// TIA Portal V21 export
FUNCTION_BLOCK "DigitalOutput"   // FB4, LAD
TITLE = FB4
{ S7_Optimized_Access := 'FALSE' }
// DIGITAL OUTPUT
// stored: AutoNumber false, SetENOAutomatically false
   VAR_INPUT
      Cmd { ExternalVisible := 'False'} : Bool;
      SimulationOn { ExternalVisible := 'False'} : Bool;
      MotorFeedbackInputSelection { ExternalVisible := 'False'} : Bool;
      MotorFeedbackInput { ExternalVisible := 'False'} : Bool;
      WaterSensorSelection { ExternalVisible := 'False'} : Bool;
      WaterSensorInput { ExternalVisible := 'False'} : Bool;
      AlwaysTrue : Bool;
      AlwaysFalse : Bool;
      OpenClose : Bool;   // For Valve Only
      Spare_3 : Bool;   // For Valve Only
      ValveFeedbackInputSelection { ExternalVisible := 'False'} : Bool;
      ValveFeedbackInput { ExternalVisible := 'False'} : Bool;
      Interlock : Bool;
      FBCheckDelay { ExternalVisible := 'False'} : Int;
      WSCheckDelay { ExternalVisible := 'False'} : Int;
      secs { ExternalVisible := 'False'} : Bool;
      AlarmAck { ExternalVisible := 'False'} : Bool;
      ModeSel : Bool;   // 1=Man/ 0=Auto
      Fault : Bool;
      Reset : Bool;
      spare : Bool;
      spare_1 : Bool;
      spare_2 : Bool;
   END_VAR
   VAR_OUTPUT
      Output { ExternalVisible := 'False'} : Bool;
      FeedBackTripAlarm : Bool;
      NoWaterFlowAlarm : Bool;
      LineColour : DInt;
      ValveColour : DInt;
      Mode : DInt;   // Auto=0 , Manual=1
      Status : DInt;
   END_VAR
   VAR_IN_OUT
      OpFbTrip { ExternalVisible := 'False'} : Bool;
      OpWaterSensorTrip { ExternalVisible := 'False'} : Bool;
      FBCheckActualTime { ExternalVisible := 'False'} : Int;
      WSCheckActualTime { ExternalVisible := 'False'} : Int;
   END_VAR
   VAR
      ResetBtn { S7_SetPoint := 'True'} : TON_TIME;
   END_VAR
   VAR_TEMP   // added for the SCL form of the ladder/FBD networks
      _w1 : Bool;
      _w2 : Bool;
   END_VAR
BEGIN

REGION Network 1: #Output
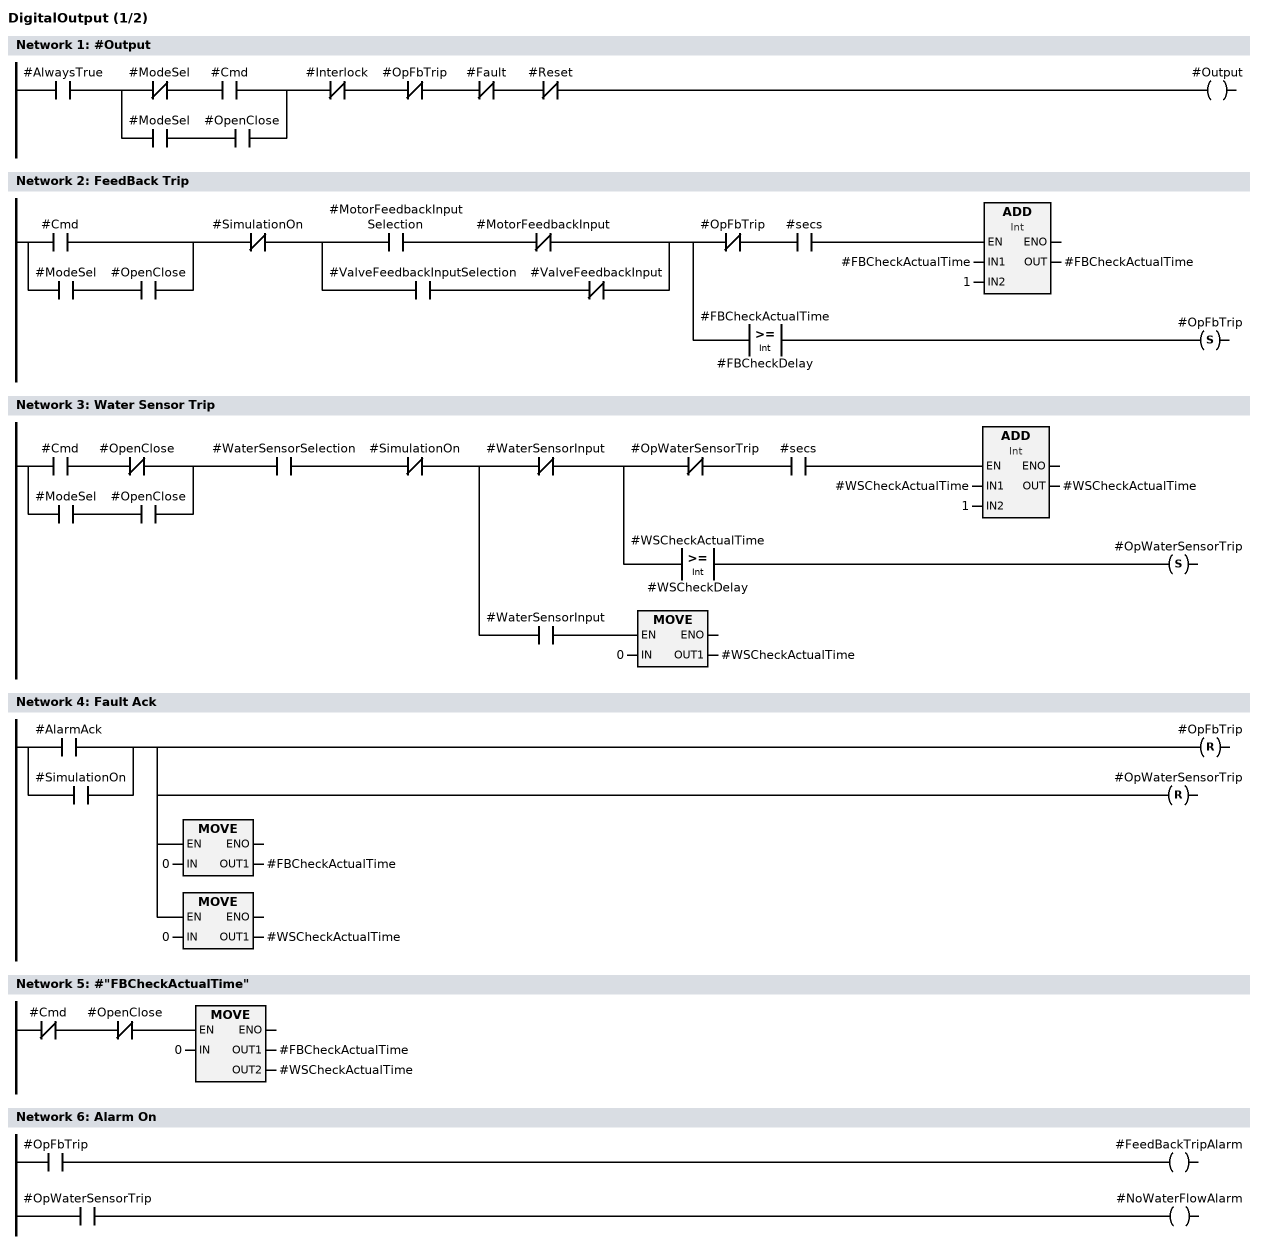
   RUNG wire#powerrail
      Contact( #AlwaysTrue )
      wire#w1
      I_Contact( #ModeSel )
      Contact( #Cmd )
      wire#w2
      I_Contact( #Interlock )
      I_Contact( #OpFbTrip )
      I_Contact( #Fault )
      I_Contact( #Reset )
      Coil( #Output )
   END_RUNG
   RUNG wire#w1
      Contact( #ModeSel )
      Contact( #OpenClose )
   END_RUNG wire#w2
   // the same network as SCL:
   #Output := #AlwaysTrue AND ((NOT #ModeSel AND #Cmd) OR (#ModeSel AND #OpenClose)) AND NOT #Interlock AND NOT #OpFbTrip AND NOT #Fault AND NOT #Reset;
END_REGION

REGION Network 2: FeedBack Trip
   RUNG wire#powerrail
      Contact( #Cmd )
      wire#w1
      I_Contact( #SimulationOn )
      wire#w2
      Contact( #MotorFeedbackInputSelection )
      I_Contact( #MotorFeedbackInput )
      wire#w3
      I_Contact( #OpFbTrip )
      Contact( #secs )
      { S7_Templates := "SrcType := Int"; S7_GenerateENO := "TRUE" } Add(in1 := #FBCheckActualTime, in2 := 1, out => #FBCheckActualTime)
   END_RUNG
   RUNG wire#powerrail
      Contact( #ModeSel )
      Contact( #OpenClose )
   END_RUNG wire#w1
   RUNG wire#w2
      Contact( #ValveFeedbackInputSelection )
      I_Contact( #ValveFeedbackInput )
   END_RUNG wire#w3
   RUNG wire#w3
      { S7_Templates := "SrcType := Int" } GE_Contact(in1 := #FBCheckActualTime, in2 := #FBCheckDelay)
      S_Coil( #OpFbTrip )
   END_RUNG
   // the same network as SCL:
   #_w1 := (#Cmd OR (#ModeSel AND #OpenClose)) AND NOT #SimulationOn AND ((#MotorFeedbackInputSelection AND NOT #MotorFeedbackInput) OR (#ValveFeedbackInputSelection AND NOT #ValveFeedbackInput));
   IF #_w1 AND NOT #OpFbTrip AND #secs THEN #FBCheckActualTime := #FBCheckActualTime + 1; END_IF;
   IF #_w1 AND (#FBCheckActualTime >= #FBCheckDelay) THEN #OpFbTrip := TRUE; END_IF;
END_REGION

REGION Network 3: Water Sensor Trip
   RUNG wire#powerrail
      Contact( #Cmd )
      I_Contact( #OpenClose )
      wire#w1
      Contact( #WaterSensorSelection )
      I_Contact( #SimulationOn )
      wire#w2
      I_Contact( #WaterSensorInput )
      wire#w3
      I_Contact( #OpWaterSensorTrip )
      Contact( #secs )
      { S7_Templates := "SrcType := Int"; S7_GenerateENO := "TRUE" } Add(in1 := #WSCheckActualTime, in2 := 1, out => #WSCheckActualTime)
   END_RUNG
   RUNG wire#powerrail
      Contact( #ModeSel )
      Contact( #OpenClose )
   END_RUNG wire#w1
   RUNG wire#w3
      { S7_Templates := "SrcType := Int" } GE_Contact(in1 := #WSCheckActualTime, in2 := #WSCheckDelay)
      S_Coil( #OpWaterSensorTrip )
   END_RUNG
   RUNG wire#w2
      Contact( #WaterSensorInput )
      { S7_GenerateENO := "TRUE" } Move(in := 0, out1 => #WSCheckActualTime)
   END_RUNG
   // the same network as SCL:
   #_w1 := ((#Cmd AND NOT #OpenClose) OR (#ModeSel AND #OpenClose)) AND #WaterSensorSelection AND NOT #SimulationOn;
   #_w2 := #_w1 AND NOT #WaterSensorInput;
   IF #_w2 AND NOT #OpWaterSensorTrip AND #secs THEN #WSCheckActualTime := #WSCheckActualTime + 1; END_IF;
   IF #_w2 AND (#WSCheckActualTime >= #WSCheckDelay) THEN #OpWaterSensorTrip := TRUE; END_IF;
   IF #_w1 AND #WaterSensorInput THEN #WSCheckActualTime := 0; END_IF;
END_REGION

REGION Network 4: Fault Ack
   RUNG wire#powerrail
      Contact( #AlarmAck )
      wire#w1
      R_Coil( #OpFbTrip )
   END_RUNG
   RUNG wire#powerrail
      Contact( #SimulationOn )
   END_RUNG wire#w1
   RUNG wire#w1
      R_Coil( #OpWaterSensorTrip )
   END_RUNG
   RUNG wire#w1
      { S7_GenerateENO := "TRUE" } Move(in := 0, out1 => #FBCheckActualTime)
   END_RUNG
   RUNG wire#w1
      { S7_GenerateENO := "TRUE" } Move(in := 0, out1 => #WSCheckActualTime)
   END_RUNG
   // the same network as SCL:
   IF #AlarmAck OR #SimulationOn THEN
       #OpFbTrip := FALSE;
       #OpWaterSensorTrip := FALSE;
       #FBCheckActualTime := 0;
       #WSCheckActualTime := 0;
   END_IF;
END_REGION

REGION Network 5: #"FBCheckActualTime"
   RUNG wire#powerrail
      I_Contact( #Cmd )
      I_Contact( #OpenClose )
      { S7_GenerateENO := "TRUE" } Move(in := 0, out1 => #FBCheckActualTime, out2 => #WSCheckActualTime)
   END_RUNG
   // the same network as SCL:
   IF NOT #Cmd AND NOT #OpenClose THEN
       #FBCheckActualTime := 0;
       #WSCheckActualTime := 0;
   END_IF;
END_REGION

REGION Network 6: Alarm On
   RUNG wire#powerrail
      Contact( #OpFbTrip )
      Coil( #FeedBackTripAlarm )
   END_RUNG
   RUNG wire#powerrail
      Contact( #OpWaterSensorTrip )
      Coil( #NoWaterFlowAlarm )
   END_RUNG
   // the same network as SCL:
   #FeedBackTripAlarm := #OpFbTrip;
   #NoWaterFlowAlarm := #OpWaterSensorTrip;
END_REGION

REGION Network 7: Valve Colour
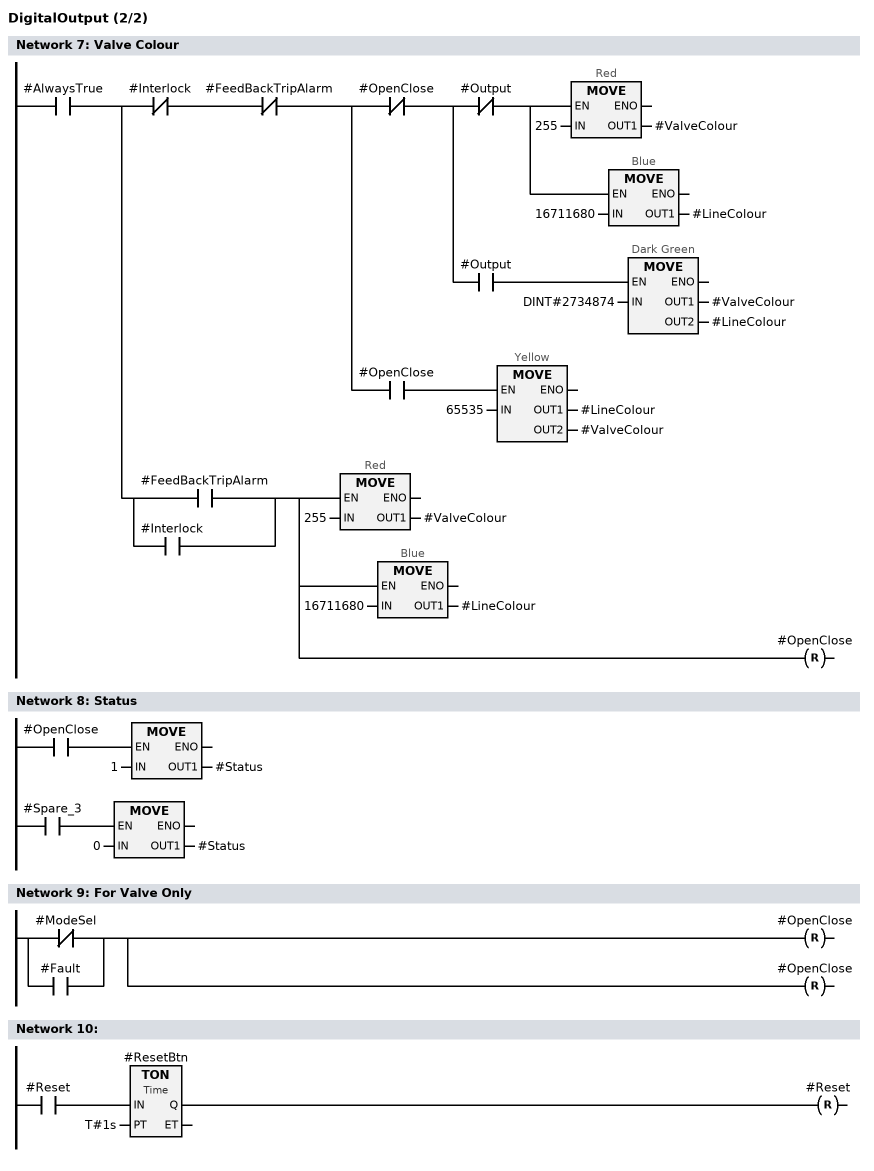
   RUNG wire#powerrail
      Contact( #AlwaysTrue )
      wire#w1
      I_Contact( #Interlock )
      I_Contact( #FeedBackTripAlarm )
      wire#w2
      I_Contact( #OpenClose )
      wire#w3
      I_Contact( #Output )
      wire#w4
      Move(in := 255, out1 => #ValveColour)   // Red
   END_RUNG
   RUNG wire#w4
      Move(in := 16711680, out1 => #LineColour)   // Blue
   END_RUNG
   RUNG wire#w3
      Contact( #Output )
      Move(in := DINT#2734874, out1 => #ValveColour, out2 => #LineColour)   // Dark Green
   END_RUNG
   RUNG wire#w2
      Contact( #OpenClose )
      Move(in := 65535, out1 => #LineColour, out2 => #ValveColour)   // Yellow
   END_RUNG
   RUNG wire#w1
      Contact( #FeedBackTripAlarm )
      wire#w5
      Move(in := 255, out1 => #ValveColour)   // Red
   END_RUNG
   RUNG wire#w1
      Contact( #Interlock )
   END_RUNG wire#w5
   RUNG wire#w5
      Move(in := 16711680, out1 => #LineColour)   // Blue
   END_RUNG
   RUNG wire#w5
      R_Coil( #OpenClose )
   END_RUNG
   // the same network as SCL:
   #_w1 := #AlwaysTrue AND NOT #Interlock AND NOT #FeedBackTripAlarm;
   #_w2 := #_w1 AND NOT #OpenClose;
   IF #_w2 AND NOT #Output THEN
       #ValveColour := 255;   // Red
       #LineColour := 16711680;   // Blue
   END_IF;
   IF #_w2 AND #Output THEN
       #ValveColour := DINT#2734874;   // Dark Green
       #LineColour := DINT#2734874;
   END_IF;
   IF #_w1 AND #OpenClose THEN
       #LineColour := 65535;   // Yellow
       #ValveColour := 65535;
   END_IF;
   IF #AlwaysTrue AND (#FeedBackTripAlarm OR #Interlock) THEN
       #ValveColour := 255;   // Red
       #LineColour := 16711680;   // Blue
       #OpenClose := FALSE;
   END_IF;
END_REGION

REGION Network 8: Status
   RUNG wire#powerrail
      Contact( #OpenClose )
      Move(in := 1, out1 => #Status)
   END_RUNG
   RUNG wire#powerrail
      Contact( #Spare_3 )
      Move(in := 0, out1 => #Status)
   END_RUNG
   // the same network as SCL:
   IF #OpenClose THEN #Status := 1; END_IF;
   IF #Spare_3 THEN #Status := 0; END_IF;
END_REGION

REGION Network 9: For Valve Only
   RUNG wire#powerrail
      I_Contact( #ModeSel )
      wire#w1
      R_Coil( #OpenClose )
   END_RUNG
   RUNG wire#powerrail
      Contact( #Fault )
   END_RUNG wire#w1
   RUNG wire#w1
      R_Coil( #OpenClose )
   END_RUNG
   // the same network as SCL:
   IF NOT #ModeSel OR #Fault THEN
       #OpenClose := FALSE;
       #OpenClose := FALSE;
   END_IF;
END_REGION

REGION Network 10
   RUNG wire#powerrail
      Contact( #Reset )
      { S7_Templates := "time_type := Time" } #ResetBtn.TON(pt := T#1s, et =>)
      R_Coil( #Reset )
   END_RUNG
   // the same network as SCL:
   #ResetBtn(IN := #Reset, PT := T#1s);   // TON
   IF #ResetBtn.Q THEN #Reset := FALSE; END_IF;
END_REGION
END_FUNCTION_BLOCK
